KUKA KRL program: arc_start_stop.src, arc_start_stop.dat

--- arc_start_stop.src ---
&ACCESS RVO2
&REL 2
&PARAM DISKPATH = KRC:\R1
DEF arc_start_stop()

END

;() 12 34

DEFFCT E6POS get_z_offset_point(offset_mm :IN)
   DECL REAL offset_mm
   DECL E6POS z_off
   z_off = $pos_act_mes
   z_off.Z = z_off.Z + offset_mm
   RETURN z_off
ENDFCT

GLOBAL DEF ARC_START_JOB(jobNumber :IN)
   ; jobNumber specifies the welding job to activate
   DECL INT jobNumber

   WDAT_VAR.Weld.Channel1 = jobNumber ; Update the specific variable

   ArcMainNG(#PreDefinition, WDAT_VAR, WP1)
   ArcMainNG(#GasPreflow, WDAT_VAR, WP1)
   ArcMainNG(#ArcOnMoveStd, WDAT_VAR, WP1)     ; Start the arc
   ArcMainNG(#ArcOnBeforeMoveStd, WDAT_VAR, WP1)
   LIN get_z_offset_point(1.2) C_VEL
   ArcMainNG(#ArcOnAfterMoveStd, WDAT_VAR, WP1)

END

GLOBAL DEF ARC_SWI_JOB(jobNumber :IN)

   ; jobNumber specifies the welding job to activate
   DECL INT jobNumber
   WDAT_VAR.Weld.Channel1 = jobNumber ; Update the specific variable

   ArcMainNG(#ArcSwiMoveStd, WDAT_VAR, WP1)

   ArcMainNG(#ArcSwiBeforeMoveStd, WDAT_VAR, WP1)
   ; LIN get_z_offset_point(1.2) C_VEL
   ArcMainNG(#ArcSwiAfterMoveStd, WDAT_VAR, WP1)

END



GLOBAL DEF ARC_STOP()
   ; copied from end of ARC start?
   ; ArcMainNG(#ArcOnAfterMoveStd, WDAT_VAR, WP1)

   ArcMainNG(#ArcOffMoveStd, WDAT_VAR, WP1)
END


GLOBAL DEF ARC_STOP_FULL()
   ArcMainNG(#ArcOffBeforeOffStd, WDAT_VAR, WP1)
   ArcMainNG(#ArcOffBeforeOffStd2, WDAT_VAR, WP1)
   ArcMainNG(#ArcOffMoveStd, WDAT_VAR, WP1)
   ArcMainNG(#ArcOffBeforeMoveStd, WDAT_VAR, WP1)
   LIN get_z_offset_point(1.2) C_VEL
   ArcMainNG(#ArcOffAfterMoveStd, WDAT_VAR, WP1)
END

--- arc_start_stop.dat ---
&ACCESS RVO2
&REL 3
&PARAM DISKPATH = KRC:\R1
DEFDAT  ARC_START_STOP PUBLIC
;; YO
;; job 17  7
;; heyo

DECL GLOBAL stArcDat_T WDAT_VAR={WdatId[] "WDAT1",Info {Version 306020371,WId 1,WName[] "Fronius TPSi job mode"},Strike {JobModeId[] "Job mode",StartTime 0.0,PreFlowTime 0.0,Channel1 0.0,Channel2 0.0,Channel3 0.0,Channel4 0.0,Channel5 0.0,Channel6 0.0,Channel7 0.0,Channel8 0.0,PurgeTime 0.0},Weld {JobModeId[] "Job mode",ParamSetId[] "Set1",Velocity 0.01000000,Channel1 5.00000,Channel2 0.0,Channel3 0.0,Channel4 0.0,Channel5 0.0,Channel6 0.0,Channel7 0.0,Channel8 0.0},Weave {Pattern #None,Length 4.00000,Amplitude 2.00000,Angle 0.0,Frequency 2.00000,LeftSideDelay 0.0,RightSideDelay 0.0},Crater {JobModeId[] "Job mode",ParamSetId[] "Set2",CraterTime 0.0,PostflowTime 0.0,Channel1 1.00000,Channel2 0.0,Channel3 0.0,Channel4 0.0,Channel5 0.0,Channel6 0.0,Channel7 0.0,Channel8 0.0,BurnBackTime 0.0}}

DECL GLOBAL stArcDat_T WDAT1={WdatId[] "WDAT1",Info {Version 306020371,WId 1,WName[] "Fronius TPSi job mode"},Strike {JobModeId[] "Job mode",StartTime 0.0,PreFlowTime 0.0,Channel1 0.0,Channel2 0.0,Channel3 0.0,Channel4 0.0,Channel5 0.0,Channel6 0.0,Channel7 0.0,Channel8 0.0,PurgeTime 0.0},Weld {JobModeId[] "Job mode",ParamSetId[] "Set1",Velocity 0.01000000,Channel1 16.0000,Channel2 0.0,Channel3 0.0,Channel4 0.0,Channel5 0.0,Channel6 0.0,Channel7 0.0,Channel8 0.0},Weave {Pattern #None,Length 4.00000,Amplitude 2.00000,Angle 0.0,Frequency 2.00000,LeftSideDelay 0.0,RightSideDelay 0.0},Crater {JobModeId[] "Job mode",ParamSetId[] "Set2",CraterTime 0.0,PostflowTime 0.0,Channel1 1.00000,Channel2 0.0,Channel3 0.0,Channel4 0.0,Channel5 0.0,Channel6 0.0,Channel7 0.0,Channel8 0.0,BurnBackTime 0.0}}
DECL GLOBAL stArcDat_T WDAT2={WdatId[] "WDAT2",Info {Version 306020371,WId 1,WName[] "Fronius TPSi job mode"},Strike {JobModeId[] "Job mode",StartTime 0.0,PreFlowTime 0.0,Channel1 0.0,Channel2 0.0,Channel3 0.0,Channel4 0.0,Channel5 0.0,Channel6 0.0,Channel7 0.0,Channel8 0.0,PurgeTime 0.0},Weld {JobModeId[] "Job mode",ParamSetId[] "Set1",Velocity 0.01000000,Channel1 17.0000,Channel2 0.0,Channel3 0.0,Channel4 0.0,Channel5 0.0,Channel6 0.0,Channel7 0.0,Channel8 0.0},Weave {Pattern #None,Length 4.00000,Amplitude 2.00000,Angle 0.0,Frequency 2.00000,LeftSideDelay 0.0,RightSideDelay 0.0},Crater {JobModeId[] "Job mode",ParamSetId[] "Set2",CraterTime 0.0,PostflowTime 0.0,Channel1 2.00000,Channel2 0.0,Channel3 0.0,Channel4 0.0,Channel5 0.0,Channel6 0.0,Channel7 0.0,Channel8 0.0,BurnBackTime 0.0}}
DECL GLOBAL stArcDat_T WDAT3={WdatId[] "WDAT3",Info {Version 306020371,WId 1,WName[] "Fronius TPSi job mode"},Strike {JobModeId[] "Job mode",StartTime 0.0,PreFlowTime 0.0,Channel1 0.0,Channel2 0.0,Channel3 0.0,Channel4 0.0,Channel5 0.0,Channel6 0.0,Channel7 0.0,Channel8 0.0,PurgeTime 0.0},Weld {JobModeId[] "Job mode",ParamSetId[] "Set1",Velocity 0.01000000,Channel1 18.0000,Channel2 0.0,Channel3 0.0,Channel4 0.0,Channel5 0.0,Channel6 0.0,Channel7 0.0,Channel8 0.0},Weave {Pattern #None,Length 4.00000,Amplitude 2.00000,Angle 0.0,Frequency 2.00000,LeftSideDelay 0.0,RightSideDelay 0.0},Crater {JobModeId[] "Job mode",ParamSetId[] "Set2",CraterTime 0.0,PostflowTime 0.0,Channel1 3.00000,Channel2 0.0,Channel3 0.0,Channel4 0.0,Channel5 0.0,Channel6 0.0,Channel7 0.0,Channel8 0.0,BurnBackTime 0.0}}
;WP1
DECL GLOBAL stArcDat_T WP1={WdatId[] "WP1",Info {Version 306020371},Strike {SeamName[] " ",PartName[] " ",SeamNumber 1,PartNumber 1,DesiredLength 0.0,LengthTolNeg 0.0,LengthTolPos 0.0,LengthCtrlActive FALSE},Advanced {BitCodedRobotMark 0}}
ENDDAT
